FUNCTION_BLOCK Sequence1Task EXTENDS TcoCore.TcoTask
VAR_INPUT
	Sequence : TcoCore.ITcoSequencer;
END_VAR

(*~
	<docu>
		<summary>
			Restores this instance to the Ready state. Can be called explicitly or from within one of the restore mechanisms.
			<para>
				See also <see cref="PlcDocu.TcoCore.TcoTask.AutoRestorable()"/>
			</para>
		</summary>			
	</docu>	
~*)
METHOD Restore : ITcoRestorable
SUPER^.Restore();
THIS^.Sequence.Restore();
END_METHOD

END_FUNCTION_BLOCK

(* stored: Version 1.1.0.1, ProductVersion 3.1.4024.12
   POU Sequence1Task: Id {76616854-4b40-0388-3307-33475d014065}, SpecialFunc None
   Method Restore: Id {2232c6fe-9e30-0098-0cdd-9148e5418ad6} *)
